(* PLC project Blank Project, Blank Blank 1.0 *)
(* stored: creationDateTime 2016-05-18T21:14:07, modificationDateTime 2017-10-17T17:24:40 *)

PROGRAM Cell1
  VAR
    R1_front AT %IX0.2 : BOOL := true;
    R1_rear AT %IX0.3 : BOOL := true;
    C1_endIR AT %IX0.4 : BOOL := true;
    C1_startIR AT %IX0.5 : BOOL := true;
    Main AT %IX0.6 : BOOL := false;
    R1_fwd_motor AT %QX0.2 : BOOL := true;
    R1_bwd_motor AT %QX0.3 : BOOL := true;
    C1_motor AT %QX0.4 : BOOL := true;
  END_VAR
  VAR
    C1_working : BOOL := false;
    State1 : BOOL := false;
  END_VAR
  VAR
    State1_int AT %MD1 : DINT := 0;
  END_VAR
  VAR
    R1_in_transit : BOOL := false;
    State2 : BOOL := false;
  END_VAR
  VAR
    State2_int AT %MD3 : DINT := 0;
  END_VAR
  VAR
    R1_fwd : BOOL := false;
  END_VAR
  VAR
    R1_fwd_int AT %MD4 : DINT := 0;
  END_VAR
  VAR
    R1_bwd : BOOL := false;
  END_VAR
  VAR
    R1_bwd_int AT %MD5 : DINT := 0;
  END_VAR
  VAR
    Timer_in_transit : TON;
  END_VAR
  VAR
    jadeProg1 AT %IX0.7 : BOOL := true;
  END_VAR

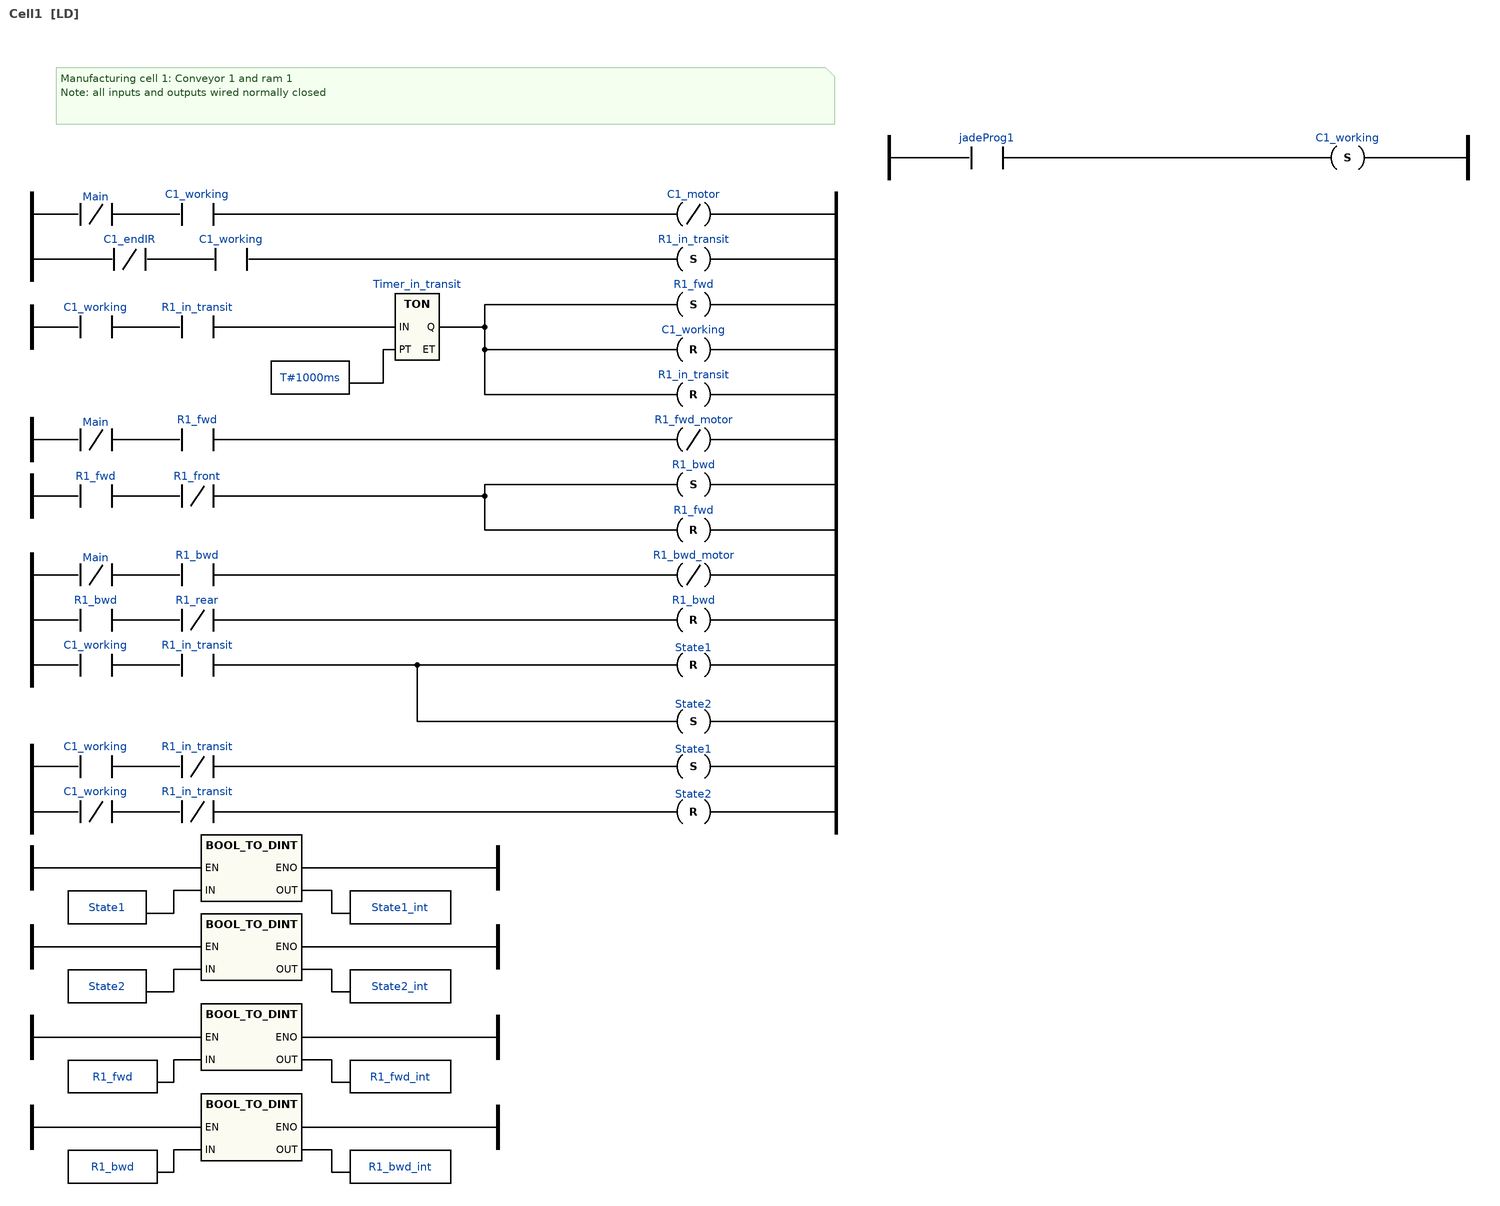
(* LD diagram, written out as Structured Text *)
(* Manufacturing cell 1: Conveyor 1 and ram 1
Note: all inputs and outputs wired normally closed *)
IF jadeProg1 THEN C1_working := TRUE; END_IF;
C1_motor := NOT (NOT Main AND C1_working);
IF NOT C1_endIR AND C1_working THEN R1_in_transit := TRUE; END_IF;
Timer_in_transit(IN := C1_working AND R1_in_transit, PT := T#1000ms);
IF Timer_in_transit.Q THEN R1_fwd := TRUE; END_IF;
IF Timer_in_transit.Q THEN C1_working := FALSE; END_IF;
IF Timer_in_transit.Q THEN R1_in_transit := FALSE; END_IF;
R1_fwd_motor := NOT (NOT Main AND R1_fwd);
IF R1_fwd AND NOT R1_front THEN R1_bwd := TRUE; END_IF;
IF R1_fwd AND NOT R1_front THEN R1_fwd := FALSE; END_IF;
R1_bwd_motor := NOT (NOT Main AND R1_bwd);
IF R1_bwd AND NOT R1_rear THEN R1_bwd := FALSE; END_IF;
IF C1_working AND R1_in_transit THEN State1 := FALSE; END_IF;
IF C1_working AND R1_in_transit THEN State2 := TRUE; END_IF;
IF C1_working AND NOT R1_in_transit THEN State1 := TRUE; END_IF;
IF NOT C1_working AND NOT R1_in_transit THEN State2 := FALSE; END_IF;
State1_int := BOOL_TO_DINT(State1);
State2_int := BOOL_TO_DINT(State2);
R1_fwd_int := BOOL_TO_DINT(R1_fwd);
R1_bwd_int := BOOL_TO_DINT(R1_bwd);
END_PROGRAM

CONFIGURATION Config0
  RESOURCE Res0 ON PLC
    TASK TaskMain(INTERVAL := T#50ms, PRIORITY := 0);
    PROGRAM Inst0 WITH TaskMain : Cell1;
  END_RESOURCE
END_CONFIGURATION
